# EPICS autosave request: iocBoot/shutter.req
$(P):SHUTTER$(N):ENABLE
$(P):SHUTTER$(N):PVNAME
$(P):SHUTTER$(N):TYPE
$(P):SHUTTER$(N):RBV
